// Hardware mapping is kept here; the machine FB has no absolute IO addresses.
PROGRAM MAIN
VAR
    machine : FB_AssemblyStation;
    command : E_ReferenceCommand;
END_VAR

machine(inputs := GVL_HW.inputs, command := command);
GVL_HW.outputs := machine.outputs;

END_PROGRAM

(* stored: Version 1.1.0.1
   POU MAIN: Id {05cb368c-66e5-4aa0-9491-7b02e519ec00}, SpecialFunc None *)
